// TIA Portal V20 export
TYPE "typeRollChangeDoor"
// stored: Access Published, IsFailsafeCompliant true, Namespace Safety
   STRUCT
      Lock : Bool;
      Unlock : Bool;
      Reset : Bool;
   END_STRUCT;
END_TYPE
